// TIA Portal V20 export
VAR_GLOBAL   // PLC tag table "Unit1Em3"
   "BA060ZSIBK06.00" AT %I1020.0 : Bool;   // TOP TAPE DIAMETER SENSOR
   "BA060ZSIBK06.01" AT %I1020.1 : Bool;   // (HOME) TOP TAPE CUTTER UP
   "BA060ZSIBK06.02" AT %I1020.2 : Bool;   // (HOME) TOP TAPE CUTTER CLAMP UP
   "BA060ZSIBK06.03" AT %I1020.3 : Bool;   // (HOME) TOP TAPE CLAMP OPEN
   "BA060ZSIBK06.04" AT %I1020.4 : Bool;   // (HOME) TOP TAPE TENSION BACKWARD
   "BA060ZSIBK06.05" AT %I1020.5 : Bool;   // (HOME) TOP TAPE LOADING BACKWARD
   "BA060ZSIBK06.06" AT %I1020.6 : Bool;   // SPARE
   "BA060ZSIBK06.07" AT %I1020.7 : Bool;   // SPARE
   "BA060ZSIBK06.08" AT %I1021.0 : Bool;   // SPARE
   "BA060ZSIBK06.09" AT %I1021.1 : Bool;   // (WORK) TOP TAPE CUTTER DOWN
   "BA060ZSIBK06.10" AT %I1021.2 : Bool;   // (WORK) TOP TAPE CUTTER CLAMP DOWN
   "BA060ZSIBK06.11" AT %I1021.3 : Bool;   // (WORK) TOP TAPE CLAMP CLOSE
   "BA060ZSIBK06.12" AT %I1021.4 : Bool;   // (WORK) TOP TAPE TENSION FORWARD
   "BA060ZSIBK06.13" AT %I1021.5 : Bool;   // (WORK) TOP TAPE LOADING FORWARD
   "BA060ZSIBK06.14" AT %I1021.6 : Bool;   // SPARE
   "BA060ZSIBK06.15" AT %I1021.7 : Bool;   // SPARE
   "BA060ZSIBK07.00" AT %I1024.0 : Bool;   // TAPE ATTACHMENT VACUUM PRESSURE SWITCH
   "BA060ZSIBK07.01" AT %I1024.1 : Bool;   // SPARE
   "BA060ZSIBK07.02" AT %I1024.2 : Bool;   // (HOME) TOP TAPE ATTACHMENT UP
   "BA060ZSIBK07.03" AT %I1024.3 : Bool;   // (WORK) TOP TAPE ATTACHMENT DOWN
   "BA060ZSIBK07.07" AT %I1024.7 : Bool;   // SPARE
   "BA060ZSIBK08.00" AT %I1028.0 : Bool;   // (HOME) TOP TAPE CLAMP TOP LEFT UP
   "BA060ZSIBK08.01" AT %I1028.1 : Bool;   // (HOME) TOP TAPE CLAMP TOP CENTER UP
   "BA060ZSIBK08.02" AT %I1028.2 : Bool;   // (HOME) TOP TAPE CLAMP TOP RIGHT UP
   "BA060ZSIBK08.03" AT %I1028.3 : Bool;   // TOP TAPE ATTACHMENT VACUUM PRESSURE SWITCH
   "BA060ZSIBK08.04" AT %I1028.4 : Bool;   // (HOME) TOP TAPE CLAMP BTM DOWN
   "BA060ZSIBK08.07" AT %I1028.7 : Bool;   // TOP TAPE FIX STAGE STACK DETECT SENSOR
   "BA060ZSIBK08.08" AT %I1029.0 : Bool;   // (WORK) TOP TAPE CLAMP TOP LEFT DOWN
   "BA060ZSIBK08.09" AT %I1029.1 : Bool;   // (WORK) TOP TAPE CLAMP TOP CENTER DOWN
   "BA060ZSIBK08.10" AT %I1029.2 : Bool;   // (WORK) TOP TAPE CLAMP TOP RIGHT DOWN
   "BA060ZSIBK08.11" AT %I1029.3 : Bool;   // SPARE
   "BA060ZSIBK08.12" AT %I1029.4 : Bool;   // (WORK) TOP TAPE CLAMP BTM UP
   "BA060ZSIBK08.14" AT %I1029.6 : Bool;   // SPARE
   "BA060ZSIBK08.15" AT %I1029.7 : Bool;   // SPARE
   "BA060ZSIPM03.00" AT %Q2008.0 : Bool;   // (HOME) TOP TAPE CUTTER UP
   "BA060ZSIPM03.01" AT %Q2008.1 : Bool;   // (WORK) TOP TAPE CUTTER DOWN
   "BA060ZSIPM03.02" AT %Q2008.2 : Bool;   // (HOME) TOP TAPE CUTTER CLAMP UP
   "BA060ZSIPM03.03" AT %Q2008.3 : Bool;   // (WORK) TOP TAPE CUTTER CLAMP DOWN
   "BA060ZSIPM03.04" AT %Q2008.4 : Bool;   // (HOME) TOP TAPE LOADING CLAMP OPEN
   "BA060ZSIPM03.05" AT %Q2008.5 : Bool;   // (WORK) TOP TAPE LOADING CLAMP CLOSE
   "BA060ZSIPM03.06" AT %Q2008.6 : Bool;   // (WORK) TOP TAPE TENSION FORWARD
   "BA060ZSIPM03.07" AT %Q2008.7 : Bool;   // (HOME) TOP TAPE TENSION BACKWARD
   "BA060ZSIPM03.10" AT %Q2009.0 : Bool;   // (WORK) TOP TAPE LOADING FORWARD
   "BA060ZSIPM03.11" AT %Q2009.1 : Bool;   // (HOME) TOP TAPE LOADING BACKWARD
   "BA060ZSIPM03.12" AT %Q2009.2 : Bool;   // (HOME) TOP TAPE ATTACHMENT UP
   "BA060ZSIPM03.13" AT %Q2009.3 : Bool;   // (WORK) TOP TAPE ATTACHMENT DOWN
   "BA060ZSIPM03.14" AT %Q2009.4 : Bool;   // SPARE
   "BA060ZSIPM03.15" AT %Q2009.5 : Bool;   // SPARE
   "BA060ZSIPM03.16" AT %Q2009.6 : Bool;   // SPARE
   "BA060ZSIPM03.17" AT %Q2009.7 : Bool;   // SPARE
   "BA060ZSIPM04.00" AT %Q2012.0 : Bool;   // (HOME) TOP TAPE Clamp TOP LEFT UP
   "BA060ZSIPM04.01" AT %Q2012.1 : Bool;   // (WORK) TOP TAPE Clamp TOP LEFT DOWN
   "BA060ZSIPM04.02" AT %Q2012.2 : Bool;   // (HOME) TOP TAPE Clamp TOP CENTER UP
   "BA060ZSIPM04.03" AT %Q2012.3 : Bool;   // (WORK) TOP TAPE Clamp TOP CENTER DOWN
   "BA060ZSIPM04.04" AT %Q2012.4 : Bool;   // (HOME) TOP TAPE Clamp TOP RIGHT UP
   "BA060ZSIPM04.05" AT %Q2012.5 : Bool;   // (WORK) TOP TAPE Clamp TOP RIGHT DOWN
   "BA060ZSIPM04.06" AT %Q2012.6 : Bool;   // (WORK) TOP TAPE Clamp BTM UP
   "BA060ZSIPM04.07" AT %Q2012.7 : Bool;   // (HOME) TOP TAPE Clamp BTM DOWN
   "BA060ZSIPM04.10" AT %Q2013.0 : Bool;   // SPARE
   "BA060ZSIPM04.11" AT %Q2013.1 : Bool;   // SPARE
   "BA060ZSIPM04.12" AT %Q2013.2 : Bool;   // SPARE
   "BA060ZSIPM04.13" AT %Q2013.3 : Bool;   // SPARE
   "BA060ZSIPM04.14" AT %Q2013.4 : Bool;   // SPARE
   "BA060ZSIPM04.15" AT %Q2013.5 : Bool;   // SPARE
   "BA060ZSIPM04.16" AT %Q2013.6 : Bool;   // SPARE
   "BA060ZSIPM04.17" AT %Q2013.7 : Bool;   // SPARE
   "BA060ZSIBK25.00" AT %Q2104.0 : Bool;   // TOP TAPE ATTACHMENT #1 VACUUM ON
   "BA060ZSIBK25.01" AT %Q2104.1 : Bool;   // TOP TAPE ATTACHMENT #1 VACUUM OFF
   "BA060ZSIBK25.02" AT %Q2104.2 : Bool;   // SPARE
   "BA060ZSIBK25.03" AT %Q2104.3 : Bool;   // SPARE
   "BA060ZSIBK25.04" AT %Q2104.4 : Bool;   // SPARE
   "BA060ZSIBK25.05" AT %Q2104.5 : Bool;   // SPARE
   "BA060ZSIBK25.06" AT %Q2104.6 : Bool;   // SPARE
   "BA060ZSIBK25.07" AT %Q2104.7 : Bool;   // SPARE
END_VAR
VAR_GLOBAL CONSTANT   // user constants
   U1EM3_JOB01 : DInt := 1;
   U1EM3_JOB02 : DInt := 2;
   U1EM3_JOB03 : DInt := 3;
   U1EM3_JOB04 : DInt := 4;
   U1EM3_JOB05 : DInt := 5;
   U1EM3_JOB06 : DInt := 6;
   U1EM3_JOB07 : DInt := 7;
   U1EM3_JOB08 : DInt := 8;
   U1EM3_JOB09 : DInt := 9;
   U1EM3_JOB10 : DInt := 10;
   U1EM3_JOB11 : DInt := 11;
   U1EM3_JOB12 : DInt := 12;
   U1EM3_JOB13 : DInt := 13;
   U1EM3_JOB14 : DInt := 14;
   U1EM3_JOB15 : DInt := 15;
   U1EM3_JOB16 : DInt := 16;
   U1EM3_JOB17 : DInt := 17;
   U1EM3_JOB18 : DInt := 18;
   U1EM3_JOB19 : DInt := 19;
   U1EM3_JOB20 : DInt := 20;
   U1EM3_JOB21 : DInt := 21;
   U1EM3_JOB22 : DInt := 22;
   U1EM3_JOB23 : DInt := 23;
   U1EM3_JOB24 : DInt := 24;
   U1EM3_JOB25 : DInt := 25;
   U1EM3_JOB26 : DInt := 26;
   U1EM3_JOB27 : DInt := 27;
   U1EM3_JOB28 : DInt := 28;
   U1EM3_JOB29 : DInt := 29;
   U1EM3_JOB30 : DInt := 30;
   U1EM3_JOB31 : DInt := 31;
   U1EM3_JOB32 : DInt := 32;
   U1EM3_JOB33 : DInt := 33;
   U1EM3_JOB34 : DInt := 34;
   U1EM3_JOB35 : DInt := 35;
   U1EM3_JOB36 : DInt := 36;
   U1EM3_JOB37 : DInt := 37;
   U1EM3_JOB38 : DInt := 38;
   U1EM3_JOB39 : DInt := 39;
   U1EM3_JOB40 : DInt := 40;
   U1EM3_JOB41 : DInt := 41;
   U1EM3_JOB42 : DInt := 42;
   U1EM3_JOB43 : DInt := 43;
   U1EM3_JOB44 : DInt := 44;
   U1EM3_JOB45 : DInt := 45;
   U1EM3_JOB46 : DInt := 46;
   U1EM3_JOB47 : DInt := 47;
   U1EM3_JOB48 : DInt := 48;
   U1EM3_JOB49 : DInt := 49;
   U1EM3_JOB50 : DInt := 50;
   U1EM3_JOB51 : DInt := 51;
   U1EM3_JOB52 : DInt := 52;
   U1EM3_JOB53 : DInt := 53;
   U1EM3_JOB54 : DInt := 54;
   U1EM3_JOB55 : DInt := 55;
   U1EM3_JOB56 : DInt := 56;
   U1EM3_JOB57 : DInt := 57;
   U1EM3_JOB58 : DInt := 58;
   U1EM3_JOB59 : DInt := 59;
   U1EM3_JOB60 : DInt := 60;
   U1EM3_JOB61 : DInt := 61;
   U1EM3_JOB62 : DInt := 62;
   U1EM3_JOB63 : DInt := 63;
   U1EM3_JOB64 : DInt := 64;
   U1EM3_JOB65 : DInt := 65;
   U1EM3_JOB66 : DInt := 66;
   U1EM3_JOB67 : DInt := 67;
   U1EM3_JOB68 : DInt := 68;
   U1EM3_JOB69 : DInt := 69;
   U1EM3_JOB70 : DInt := 70;
   U1EM3_JOB71 : DInt := 71;
   U1EM3_JOB72 : DInt := 72;
   U1EM3_JOB73 : DInt := 73;
   U1EM3_JOB74 : DInt := 74;
   U1EM3_JOB75 : DInt := 75;
   U1EM3_JOB76 : DInt := 76;
   U1EM3_JOB77 : DInt := 77;
   U1EM3_JOB78 : DInt := 78;
   U1EM3_JOB79 : DInt := 79;
   U1EM3_JOB80 : DInt := 80;
   U1EM3_JOB81 : DInt := 81;
   U1EM3_JOB82 : DInt := 82;
   U1EM3_JOB83 : DInt := 83;
   U1EM3_JOB84 : DInt := 84;
   U1EM3_JOB85 : DInt := 85;
   U1EM3_JOB86 : DInt := 86;
   U1EM3_JOB87 : DInt := 87;
   U1EM3_JOB88 : DInt := 88;
   U1EM3_JOB89 : DInt := 89;
   U1EM3_JOB90 : DInt := 90;
   U1EM3_JOB91 : DInt := 91;
   U1EM3_JOB92 : DInt := 92;
   U1EM3_JOB93 : DInt := 93;
   U1EM3_JOB94 : DInt := 94;
   U1EM3_JOB95 : DInt := 95;
   U1EM3_JOB96 : DInt := 96;
   U1EM3_JOB97 : DInt := 97;
   U1EM3_JOB98 : DInt := 98;
   U1EM3_JOB99 : DInt := 99;
   U1EM3_SEQUENCE01 : Int := 1;
   U1EM3_SEQUENCE02 : Int := 2;
   U1EM3_SEQUENCE03 : Int := 3;
   U1EM3_SEQUENCE04 : Int := 4;
   U1EM3_SEQUENCE05 : Int := 5;
   U1EM3_SEQUENCE06 : Int := 6;
   U1EM3_SEQUENCE07 : Int := 7;
   U1EM3_SEQUENCE08 : Int := 8;
   U1EM3_SEQUENCE09 : Int := 9;
   U1EM3_SEQUENCE10 : Int := 10;
   U1EM3_SEQUENCE11 : Int := 11;
   U1EM3_SEQUENCE12 : Int := 12;
   U1EM3_SEQUENCE13 : Int := 13;
   U1EM3_SEQUENCE14 : Int := 14;
   U1EM3_SEQUENCE15 : Int := 15;
   U1EM3_SEQUENCE16 : Int := 16;
   U1EM3_SEQUENCE17 : Int := 17;
   U1EM3_SEQUENCE18 : Int := 18;
   U1EM3_SEQUENCE19 : Int := 19;
   U1EM3_SEQUENCE20 : Int := 20;
   U1EM3_SEQUENCE21 : Int := 21;
   U1EM3_SEQUENCE22 : Int := 22;
   U1EM3_SEQUENCE23 : Int := 23;
   U1EM3_SEQUENCE24 : Int := 24;
   U1EM3_SEQUENCE25 : Int := 25;
   U1EM3_SEQUENCE26 : Int := 26;
   U1EM3_SEQUENCE27 : Int := 27;
   U1EM3_SEQUENCE28 : Int := 28;
   U1EM3_SEQUENCE29 : Int := 29;
   U1EM3_SEQUENCE30 : Int := 30;
   U1EM3_SEQUENCE31 : Int := 31;
   U1EM3_SEQUENCE32 : Int := 32;
   U1EM3_SEQUENCE33 : Int := 33;
   U1EM3_SEQUENCE34 : Int := 34;
   U1EM3_SEQUENCE35 : Int := 35;
   U1EM3_SEQUENCE36 : Int := 36;
   U1EM3_SEQUENCE37 : Int := 37;
   U1EM3_SEQUENCE38 : Int := 38;
   U1EM3_SEQUENCE39 : Int := 39;
   U1EM3_SEQUENCE40 : Int := 40;
   U1EM3_SEQUENCE41 : Int := 41;
   U1EM3_SEQUENCE42 : Int := 42;
   U1EM3_SEQUENCE43 : Int := 43;
   U1EM3_SEQUENCE44 : Int := 44;
   U1EM3_SEQUENCE45 : Int := 45;
   U1EM3_SEQUENCE46 : Int := 46;
   U1EM3_SEQUENCE47 : Int := 47;
   U1EM3_SEQUENCE48 : Int := 48;
   U1EM3_SEQUENCE49 : Int := 49;
   U1EM3_SEQUENCE50 : Int := 50;
   U1EM3_SEQUENCE51 : Int := 51;
   U1EM3_SEQUENCE52 : Int := 52;
   U1EM3_SEQUENCE53 : Int := 53;
   U1EM3_SEQUENCE54 : Int := 54;
   U1EM3_SEQUENCE55 : Int := 55;
   U1EM3_SEQUENCE56 : Int := 56;
   U1EM3_SEQUENCE57 : Int := 57;
   U1EM3_SEQUENCE58 : Int := 58;
   U1EM3_SEQUENCE59 : Int := 59;
   U1EM3_SEQUENCE60 : Int := 60;
   U1EM3_SEQUENCE61 : Int := 61;
   U1EM3_SEQUENCE62 : Int := 62;
   U1EM3_SEQUENCE63 : Int := 63;
   U1EM3_SEQUENCE64 : Int := 64;
   U1EM3_SEQUENCE65 : Int := 65;
   U1EM3_SEQUENCE66 : Int := 66;
   U1EM3_SEQUENCE67 : Int := 67;
   U1EM3_SEQUENCE68 : Int := 68;
   U1EM3_SEQUENCE69 : Int := 69;
   U1EM3_SEQUENCE70 : Int := 70;
   U1EM3_SEQUENCE71 : Int := 71;
   U1EM3_SEQUENCE72 : Int := 72;
   U1EM3_SEQUENCE73 : Int := 73;
   U1EM3_SEQUENCE74 : Int := 74;
   U1EM3_SEQUENCE75 : Int := 75;
   U1EM3_SEQUENCE76 : Int := 76;
   U1EM3_SEQUENCE77 : Int := 77;
   U1EM3_SEQUENCE78 : Int := 78;
   U1EM3_SEQUENCE79 : Int := 79;
   U1EM3_SEQUENCE80 : Int := 80;
   U1EM3_SEQUENCE81 : Int := 81;
   U1EM3_SEQUENCE82 : Int := 82;
   U1EM3_SEQUENCE83 : Int := 83;
   U1EM3_SEQUENCE84 : Int := 84;
   U1EM3_SEQUENCE85 : Int := 85;
   U1EM3_SEQUENCE86 : Int := 86;
   U1EM3_SEQUENCE87 : Int := 87;
   U1EM3_SEQUENCE88 : Int := 88;
   U1EM3_SEQUENCE89 : Int := 89;
   U1EM3_SEQUENCE90 : Int := 90;
   U1EM3_SEQUENCE91 : Int := 91;
   U1EM3_SEQUENCE92 : Int := 92;
   U1EM3_SEQUENCE93 : Int := 93;
   U1EM3_SEQUENCE94 : Int := 94;
   U1EM3_SEQUENCE95 : Int := 95;
   U1EM3_SEQUENCE96 : Int := 96;
   U1EM3_SEQUENCE97 : Int := 97;
   U1EM3_SEQUENCE98 : Int := 98;
   U1EM3_SEQUENCE99 : Int := 99;
   U1EM3_NO_OF_SEQUENCE : USInt := 3;
   U1EM3_NO_OF_AXES : USInt := 2;
END_VAR
